FUNCTION_BLOCK FB_Syntax_PropertySet
VAR
    _nStored : INT;
END_VAR

_nStored := P_Value;

PROPERTY P_Value : INT
GET
P_Value := _nStored;
END_GET
SET
_nStored := P_Value;
END_SET
END_PROPERTY

END_FUNCTION_BLOCK

(* stored: Version 1.1.0.1, ProductVersion 3.1.4024.16
   POU FB_Syntax_PropertySet: Id {0da76f9d-fcd6-4b45-962b-5e428c160940}, SpecialFunc None
   Property P_Value: Id {6bc720a5-6e9b-40f5-9aa3-74319d8a2df7}
   Get Get: Id {a7246a3f-003f-483b-bdac-db32ed8111a3}
   Set Set: Id {50e7ded3-9b05-483f-b0de-99dc831afe71} *)
